// TIA Portal V20 export
FUNCTION_BLOCK "LER_CheckCamRecipeChanged"   // FB154, SCL
// stored: Access Published, MemoryReserve 100, SetENOAutomatically false
   VAR_INPUT
      calculateCamDone : Bool;   // Cam calculation Done feedback mapped from the unit DB
      unitRecipe : "typeUnitRecipe";   // Current unit recipe values used for cam calculation
      stack1UnUse : Bool;   // TRUE when Stack1 is not used for cam calculation
      stack2UnUse : Bool;   // TRUE when Stack2 is not used for cam calculation
   END_VAR
   VAR_OUTPUT
      ValidParameters : Bool;   // TRUE when monitored cam recipe values are within the allowed range
      ParameterChanged : Bool;   // TRUE when current cam recipe values differ from the last completed calculation snapshot
      ExecuteRequired : Bool;   // Latched request signal for cam calculation Execute until a fresh Done is received
   END_VAR
   VAR
      statInitialized : Bool;   // TRUE after the first completed calculation snapshot is stored
      statActive : Bool;   // Internal latch while automatic recalculation is requested or running
      statDoneArmed : Bool;   // Arms completion detection after Done has gone low
      statLastCalculatedRecipe : "typeUnitRecipe";   // Cam recipe snapshot from the last completed calculation
      statLastCalculatedStack1UnUse : Bool;   // Stack1 use state snapshot from the last completed calculation
      statLastCalculatedStack2UnUse : Bool;   // Stack2 use state snapshot from the last completed calculation
   END_VAR
BEGIN
   REGION ValidateRecipe
       // Check only the recipe values used by cam calculation.
       #ValidParameters :=
           (#unitRecipe.CPM > 0.0) AND
           (#unitRecipe.electrodWidth > 0.0) AND
           (#unitRecipe.TabSensorToCutterDistance >= 0.0) AND
           (#unitRecipe.TabSensorToCutterDistanceOffset >= 0.0) AND
           (#unitRecipe.TapeSensorToCutDistance >= 0.0) AND
           (#unitRecipe.CutToVisionSensorDistance >= 0.0) AND
           (#unitRecipe.CutToNgKickerDistance >= 0.0);
   END_REGION

   REGION CompleteRecalculation
        // Accept completion only after stale Done has cleared.
        IF #statActive THEN
            IF NOT #calculateCamDone THEN
                #statDoneArmed := TRUE;
            END_IF;

            IF #statDoneArmed AND #calculateCamDone THEN
                #statLastCalculatedRecipe := #unitRecipe;
                #statLastCalculatedStack1UnUse := #stack1UnUse;
                #statLastCalculatedStack2UnUse := #stack2UnUse;
                #statInitialized := TRUE;
                #statActive := FALSE;
                #statDoneArmed := FALSE;
            END_IF;
        END_IF;
    END_REGION

    REGION DetectRecipeChange
        // Compare the current recipe with the last completed calculation snapshot.
        #ParameterChanged :=
            (NOT #statInitialized) OR
            (#unitRecipe.CPM <> #statLastCalculatedRecipe.CPM) OR
            (#unitRecipe.electrodWidth <> #statLastCalculatedRecipe.electrodWidth) OR
            (#unitRecipe.electrodTabWidth <> #statLastCalculatedRecipe.electrodTabWidth) OR
            (#unitRecipe.electrodTabToEdge <> #statLastCalculatedRecipe.electrodTabToEdge) OR
            (#unitRecipe.electrodeGapWidth <> #statLastCalculatedRecipe.electrodeGapWidth) OR
            (#unitRecipe.electrodeThickness <> #statLastCalculatedRecipe.electrodeThickness) OR
            (#unitRecipe.TabSensorToCutterDistance <> #statLastCalculatedRecipe.TabSensorToCutterDistance) OR
            (#unitRecipe.TabSensorToCutterDistanceOffset <> #statLastCalculatedRecipe.TabSensorToCutterDistanceOffset) OR
            (#unitRecipe.TapeSensorToCutDistance <> #statLastCalculatedRecipe.TapeSensorToCutDistance) OR
            (#unitRecipe.CutToVisionSensorDistance <> #statLastCalculatedRecipe.CutToVisionSensorDistance) OR
            (#unitRecipe.CutToNgKickerDistance <> #statLastCalculatedRecipe.CutToNgKickerDistance) OR
            (#unitRecipe.CutConveyorOffset <> #statLastCalculatedRecipe.CutConveyorOffset) OR
            (#unitRecipe.NGConveyorOffset <> #statLastCalculatedRecipe.NGConveyorOffset) OR
            (#unitRecipe.Stack1ConveyorOffset <> #statLastCalculatedRecipe.Stack1ConveyorOffset) OR
            (#unitRecipe.Stack2ConveyorOffset <> #statLastCalculatedRecipe.Stack2ConveyorOffset) OR
            (#stack1UnUse <> #statLastCalculatedStack1UnUse) OR
            (#stack2UnUse <> #statLastCalculatedStack2UnUse);
    END_REGION

    REGION CancelRecalculation
        // Drop a pending request when the current values return to the last calculated snapshot.
        IF #statActive AND NOT #ParameterChanged THEN
            #statActive := FALSE;
            #statDoneArmed := FALSE;
        END_IF;
    END_REGION

    REGION RequestRecalculation
        // Latch a recalculation request while current values differ from the last completed snapshot.
        IF #ValidParameters AND #ParameterChanged AND NOT #statActive THEN
            #statActive := TRUE;
            #statDoneArmed := FALSE;
        END_IF;
    END_REGION

    REGION UpdateOutputs
        // Keep ExecuteRequired TRUE while a recalculation request is active.
        #ExecuteRequired := #statActive;
    END_REGION
END_FUNCTION_BLOCK
